TYPE T_CoESubIndex : BYTE; END_TYPE

(* stored: Version 1.1.0.1, ProductVersion 3.1.4024.14
   DUT T_CoESubIndex: Id {40c1e43a-7669-0383-2633-e7c3eab7ff62} *)
